FUNCTION_BLOCK RAWSTRING2RAWSTRING (* Basic Function Block Type *)
  (* Standard: 61499-2 *)
  (* Version 0.0, 2015-11-05, 4DIAC-IDE, 4DIAC-Consortium *)
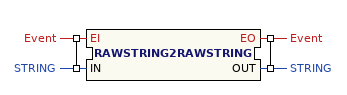
  EVENT_INPUT
    EI WITH IN;
  END_EVENT
  EVENT_OUTPUT
    EO WITH OUT;
  END_EVENT
  VAR_INPUT
    IN : STRING;
  END_VAR
  VAR_OUTPUT
    OUT : STRING;
  END_VAR
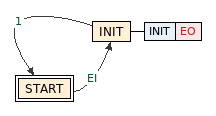
  EC_STATES
    START; (* Initial State *)
    INIT : INIT -> EO; (* Initialization *)
  END_STATES
  EC_TRANSITIONS
    START TO INIT := EI;
    INIT TO START := 1;
  END_TRANSITIONS
  ALGORITHM INIT IN ST: (* Initialization algorithm *)
IN:=OUT;
  END_ALGORITHM
END_FUNCTION_BLOCK
